// TwinCAT 3 PLC project Main
// ProgramVersion: 3.1.4023.0
// libraries:
//   Tc2_Standard, * (Beckhoff Automation GmbH)
//   Tc2_System, * (Beckhoff Automation GmbH)
//   Tc2_Utilities, * (Beckhoff Automation GmbH)
//   Tc3_Module, * (Beckhoff Automation GmbH)
// project tree:
//   / PlcTask.TcTTO
//   POUs/ MAIN.TcPOU
// real-time tasks:
//   TASK PlcTask: cycle T#10ms, priority 20, ADS port 350

CONFIGURATION Main
    RESOURCE PLC ON TwinCAT3
        TASK PlcTask(INTERVAL := T#10ms, PRIORITY := 20);
        PROGRAM MAIN WITH PlcTask : MAIN;
    END_RESOURCE
END_CONFIGURATION

// ---- POUs/MAIN.TcPOU
PROGRAM MAIN
VAR
	sizeRemaining : LINT := -1;
	start : BOOL;
	ntStart : NT_StartProcess;
END_VAR

ntStart(
	NetId := '',
	PathStr := 'C:\Windows\System32\mshta vbscript:Execute("CreateObject(""WScript.Shell"").Run ""powershell -c $$A=Get-Volume -DriveLetter C;$$B=get-adsroute -local;$$C=New-TcSession -Route $$B -Port 851;',
	DirName := 'C:\Windows\System32',
	ComndLine := 'Write-TcValue -Session $$C -Path $'Main.sizeRemaining$' -value $$A.SizeRemaining -Force;Close-TcSession -InputObject $$C;"", 0: window.close")',
	Start := start,
	TmOut := DEFAULT_ADS_TIMEOUT
);

IF start THEN
	sizeRemaining := -1;
	start := FALSE;
END_IF

END_PROGRAM
